TYPE BaseConfiguration :
STRUCT
	sName : STRING;
	sOutputDescription : STRING;
	sMountingPoint : STRING;
END_STRUCT
END_TYPE

(* stored: Version 1.1.0.1, ProductVersion 3.1.4024.9
   DUT BaseConfiguration: Id {f61b4437-cd69-45a7-b039-cc361cfd0bce} *)
